FUNCTION_BLOCK AW_EQ (* equal (IN1 = IN2 = TRUE) *)
  (* Standard: 61131-3; Classification: standard comparison function; Description: Copyright (c) 2013 TU Wien ACIN This program and the accompanying materials are made available under the terms of the Eclipse Public License 2.0 which is available at https://www.eclipse.org/legal/epl-2.0/ SPDX-License-Identifier: EPL-2.0 *)
  (* Version 3.0, 2025-04-14, Patrick Aigner, changed package *)
  (* Version 1.0, 2013-03-13, Monika Wenger, TU Wien ACIN *)
  (* Version 1.1, 2026-08-13, Franz Höpfinger, HR Agrartechnik GmbH, extended comparison family to all adapter types *)
  PACKAGE adapter::iec61131::comparison;
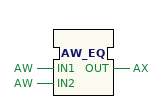
  SOCKETS
    IN1 : adapter::types::unidirectional::AW; (* Input value 1 -- left operand (IN1 = IN2) *)
    IN2 : adapter::types::unidirectional::AW; (* Input value 2 -- right operand (IN1 = IN2) *)
  END_SOCKETS
  PLUGS
    OUT : adapter::types::unidirectional::AX; (* IN1 = IN2 = TRUE *)
  END_PLUGS
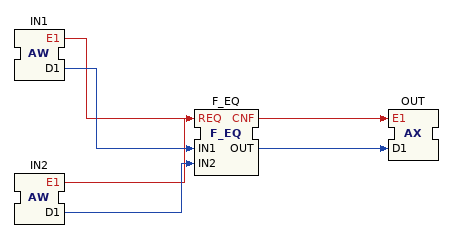
  FBS
    F_EQ : iec61131::comparison::F_EQ;
  END_FBS
  EVENT_CONNECTIONS
    F_EQ.CNF TO OUT.E1;
    IN1.E1 TO F_EQ.REQ;
    IN2.E1 TO F_EQ.REQ;
  END_CONNECTIONS
  DATA_CONNECTIONS
    F_EQ.OUT TO OUT.D1;
    IN1.D1 TO F_EQ.IN1;
    IN2.D1 TO F_EQ.IN2;
  END_CONNECTIONS
END_FUNCTION_BLOCK
